// TIA Portal V16 export
// export: Created 2024-06-17T18:37:12.7488597Z, ExportSetting WithDefaults, DisplayName Totally Integrated Automation Portal, DisplayVersion V16, DisplayName TIA Portal Version Control Interface, DisplayVersion V16, DisplayName TIA Portal Openness, DisplayVersion V16, DisplayName STEP 7 Professional, DisplayVersion V16, DisplayName STEP 7 Safety, DisplayVersion V16, DisplayName WinCC Advanced, DisplayVersion V16
TYPE "Axis.SeleçãoPainel"
// stored: IsFailsafeCompliant false
   STRUCT
      Automático : Bool;
      Manual : Bool;
      Passo_A_Passo : Bool;
      DryRun : Bool;
      IniciarCiclo : Bool;
      PararCiclo : Bool;
      VoltarPassoAnt : Bool;
      PularPassoAtual : Bool;
      ResetPassos : Bool;
      ResetFalhas : Bool;
      Liga_Comando : Bool;
   END_STRUCT;
END_TYPE
